// TwinCAT 3 PLC project PLC_1
// ProgramVersion: 3.1.4023.0
// libraries:
//   Tc2_Standard, * (Beckhoff Automation GmbH)
//   Tc2_System, * (Beckhoff Automation GmbH)
//   Tc3_Module, * (Beckhoff Automation GmbH)
// project tree:
//   / PlcTask.TcTTO
//   POUs/ FB_1.TcPOU, FB_2.TcPOU, FB_Modulo.TcPOU, MAIN.TcPOU
// real-time tasks:
//   TASK PlcTask: cycle T#10ms, priority 20, ADS port 350

CONFIGURATION PLC_1
    RESOURCE PLC ON TwinCAT3
        TASK PlcTask(INTERVAL := T#10ms, PRIORITY := 20);
        PROGRAM MAIN WITH PlcTask : MAIN;
    END_RESOURCE
END_CONFIGURATION

// ---- POUs/MAIN.TcPOU
PROGRAM MAIN
VAR
	fbAdd:		FB_1;
	fbMult:		FB_2;
	
	//New Fb
	fbDiv:		FB_Divide;
	
	nResult1:		INT;
	nResult2:		INT;
	nResult3:		INT;
END_VAR

fbAdd(nIn1:=10,
	  nIn2:=20,
	  nOut1=>nResult1);
	  
fbMult(nIn1:=10,
	  nIn2:=20,
	  nOut1=>nResult2);
	  
//New cool divide function
fbDiv(nDivIn1:=20,
	  nDivIn2:=10,
	  nDivOut=>nResult3);

END_PROGRAM

// ---- POUs/FB_1.TcPOU
//add
FUNCTION_BLOCK FB_1
VAR_INPUT
	nIn1:		INT;
	nIn2:		INT;
END_VAR
VAR_OUTPUT
	nOut1:		INT;
END_VAR
VAR
END_VAR

nOut1:=nIn1+nIn2;

END_FUNCTION_BLOCK

// ---- POUs/FB_2.TcPOU
//Multiply
FUNCTION_BLOCK FB_2
VAR_INPUT
	nIn1:		INT;
	nIn2:		INT;
END_VAR
VAR_OUTPUT
	nOut1:		INT;
END_VAR
VAR
END_VAR

nOut1:=nIn1*nIn2;

END_FUNCTION_BLOCK

// ---- POUs/FB_Modulo.TcPOU
FUNCTION_BLOCK FB_Modulo
VAR_INPUT
	fModIn1:		INT;
	fModIn2:		INT;
END_VAR
VAR_OUTPUT
	fModOut:	INT;
END_VAR
VAR
END_VAR

fModOut:= fModIn1 MOD fModIn2;

END_FUNCTION_BLOCK
